# EPICS alarm handler configuration: alh_files/mgnt_li30_lgps.alhConfig
GROUP NULL LGPS:LI30:MG01
$ALIAS LGPS
$GUIDANCE
LI30 LGPS magnets
   Group Name: LGPS:LI30:MG01
   Summary PV:  LGPS:LI30:MG01:STATSUMY
$END

GROUP LGPS:LI30:MG01  LGPS:LI30:2
CHANNEL     LGPS:LI30:2           LGPS:LI30:2:STATMSG   -----
   $FORCEPV LGPS:LI30:2:STATMSGSV -DATL 1 0
